TYPE ST_PackML_Control_Simplified :
	STRUCT
		//ClearPermissive : BOOL;
		ResetPermissive : BOOL;
		StartPermissive : BOOL;
		StopPermissive	: BOOL;
		//ClearPressed    : BOOL;
		ResetPressed : BOOL;
		StartPressed : BOOL;
		StopPressed	 : BOOL;
	END_STRUCT
END_TYPE

(* stored: Version 1.1.0.1, ProductVersion 3.1.4024.12
   DUT ST_PackML_Control_Simplified: Id {132dda0f-f204-45d3-a336-c2181759b91f} *)
